PROGRAM main
  VAR
    START_BELT : BOOL := FALSE;
    STOP_BELT : BOOL := FALSE;
    TIMER : TON;
    OBJECT_SENSOR : BOOL := FALSE;
    CONVEYOR_MOTOR : BOOL := FALSE;
    buffer : BOOL;
  END_VAR

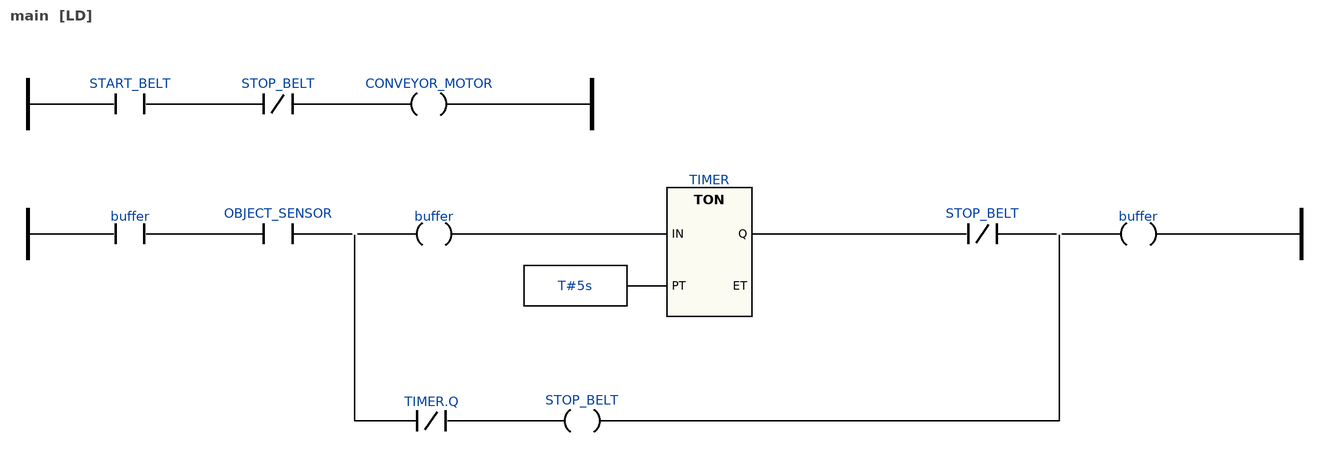
(* LD diagram, written out as Structured Text *)
CONVEYOR_MOTOR := START_BELT AND NOT STOP_BELT;
buffer := buffer AND OBJECT_SENSOR;
STOP_BELT := buffer AND OBJECT_SENSOR AND NOT TIMER.Q;
TIMER(IN := buffer AND OBJECT_SENSOR, PT := T#5s);
buffer := TIMER.Q AND NOT STOP_BELT OR buffer AND OBJECT_SENSOR AND NOT TIMER.Q;
END_PROGRAM
